(* IEC 61131-3 sources: eCockpitGit/test_project/src/%F%00 Library/%F%Common Functions/%F%Linearsation/%F%DINT, 3 files *)

(* ---- %POU%FU_diLinear2Ends.st ---- *)
//This function, converts an x, value to an y value using and 2 points on the x and y scale
//This function has ends, which means the output is never greater or smaller than the range of y
// +-----------+----------+----------+-----------------------------------------------------------------------------------------------------------------------+
// |**Version**|**Author**| **Date** |**Changes**                                                                                                            |
// +-----------+----------+----------+-----------------------------------------------------------------------------------------------------------------------+
// | 1         | NSN      | 10-12-18 | Creation                                                                                                              |
// +-----------+----------+----------+-----------------------------------------------------------------------------------------------------------------------+
FUNCTION FU_diLinear2Ends : DINT
VAR_INPUT
	XIn		:DINT;
	X1		:DINT;
	X2		:DINT;
	Y1		:DINT;
	Y2		:DINT;
END_VAR
VAR
	a		:REAL;
	b		:REAL;
END_VAR
(*%!%__DELIMITER__%!%*)
IF X2 > X1 THEN
	IF XIn <= X1 THEN	//When input is out of bounds
		FU_diLinear2Ends 			:=		Y1;
	ELSIF XIn >= X2 THEN	//When input is out of bounds
		FU_diLinear2Ends 			:=		Y2;
	ELSIF XIn > X1 AND XIn < X2 THEN	//When input is with the
		//a value is calculated
		IF X2 - X1 = 0 THEN	a := 0; ELSE a := TO_REAL(Y2 - Y1) / TO_REAL(X2 - X1); END_IF
		//b value is calculated
		b 							:=		TO_REAL(Y1) - (a * TO_REAL(X1));
		//Output is calculated
		FU_diLinear2Ends 			:=		TO_INT(a * TO_REAL (XIn) + b);
	END_IF
ELSE
	IF XIn >= X1 THEN
		FU_diLinear2Ends 			:=		Y1;
	ELSIF XIn <= X2 THEN
		FU_diLinear2Ends 			:=		Y2;
	ELSIF XIn < X1 AND XIn > X2 THEN
		//a value is calculated
		IF X2 - X1 = 0 THEN	a := 0; ELSE a := TO_REAL(Y2 - Y1) / TO_REAL(X2 - X1); END_IF
		//b value is calculated
		b 							:=		TO_REAL(Y1) - (a * TO_REAL(X1));
		//Output is calculated
		FU_diLinear2Ends 			:=		TO_INT(a * TO_REAL (XIn) + b);
	END_IF
END_IF

(* ---- %POU%FU_diLinear4Ends.st ---- *)
//This function, converts an x, value to an y value using and 3 points on the x and y scale
//This function has ends, which means the output is never greater or smaller than the range of y
// +-----------+----------+----------+-----------------------------------------------------------------------------------------------------------------------+
// |**Version**|**Author**| **Date** |**Changes**                                                                                                            |
// +-----------+----------+----------+-----------------------------------------------------------------------------------------------------------------------+
// | 1         | NSN      | 11-12-18 | Creation                                                                                                              |
// +-----------+----------+----------+-----------------------------------------------------------------------------------------------------------------------+
FUNCTION FU_diLinear4Ends : DINT
VAR_INPUT
	XIn		:DINT;
	X1		:DINT;
	X2		:DINT;
	X3		:DINT;
	X4		:DINT;
	Y1		:DINT;
	Y2		:DINT;
	Y3		:DINT;
	Y4		:DINT;
END_VAR
VAR
	a		:REAL;
	b		:REAL;
END_VAR
(*%!%__DELIMITER__%!%*)
IF X4 > X1 THEN
	IF XIn <= X1 THEN	//When input is out of bounds
		FU_diLinear4Ends 			:=		Y1;
	ELSIF XIn >= X4 THEN	//When input is out of bounds
		FU_diLinear4Ends 			:=		Y4;
	ELSIF XIn > X1 AND XIn <= X2 THEN	//When input is with the
		//a value is calculated
		IF X2 - X1 = 0 THEN	a := 0; ELSE a := TO_REAL(Y2 - Y1) / TO_REAL(X2 - X1); END_IF
		//b value is calculated
		b 							:=		TO_REAL(Y1) - (a * TO_REAL(X1));
		//Output is calculated
		FU_diLinear4Ends 			:=		TO_DINT(a * TO_REAL (XIn) + b);
	ELSIF XIn > X2 AND XIn <= X3 THEN
		//a value is calculated
		IF X3 - X2 = 0 THEN	a := 0; ELSE a := TO_REAL(Y3 - Y2) / TO_REAL(X3 - X2); END_IF
		//b value is calculated
		b 							:=		TO_REAL(Y2) - (a * TO_REAL(X2));
		//Output is calculated
		FU_diLinear4Ends 			:=		TO_INT(a * TO_REAL (XIn) + b);
	ELSIF XIn > X3 AND XIn < X4 THEN
		//a value is calculated
		IF X4 - X3 = 0 THEN	a := 0; ELSE a := TO_REAL(Y4 - Y3) / TO_REAL(X4 - X3); END_IF
		//b value is calculated
		b 							:=		TO_REAL(Y3) - (a * TO_REAL(X3));
		//Output is calculated
		FU_diLinear4Ends 			:=		TO_INT(a * TO_REAL (XIn) + b);
	END_IF
ELSE
	IF XIn >= X1 THEN
		FU_diLinear4Ends 			:=		Y1;
	ELSIF XIn <= X4 THEN
		FU_diLinear4Ends 			:=		Y4;
	ELSIF XIn < X1 AND XIn >= X2 THEN
		//a value is calculated
		IF X2 - X1 = 0 THEN	a := 0; ELSE a := TO_REAL(Y2 - Y1) / TO_REAL(X2 - X1); END_IF
		//b value is calculated
		b 							:=		TO_REAL(Y1) - (a * TO_REAL(X1));
		//Output is calculated
		FU_diLinear4Ends 			:=		TO_INT(a * TO_REAL (XIn) + b);
	ELSIF XIn < X2 AND XIn >= X3 THEN
		//a value is calculated
		IF X3 - X2 = 0 THEN	a := 0; ELSE a := TO_REAL(Y3 - Y2) / TO_REAL(X3 - X2); END_IF
		//b value is calculated
		b 							:=		TO_REAL(Y2) - (a * TO_REAL(X2));
		//Output is calculated
		FU_diLinear4Ends 			:=		TO_INT(a * TO_REAL (XIn) + b);
	ELSIF XIn < X3 AND XIn > X4 THEN
		//a value is calculated
		IF X4 - X3 = 0 THEN	a := 0; ELSE a := TO_REAL(Y4 - Y3) / TO_REAL(X4 - X3); END_IF
		//b value is calculated
		b 							:=		TO_REAL(Y3) - (a * TO_REAL(X3));
		//Output is calculated
		FU_diLinear4Ends 			:=		TO_INT(a * TO_REAL (XIn) + b);
	END_IF
END_IF

(* ---- %POU%FU_diLinearXEnds.st ---- *)
//This function, converts an x, value to an y value using and x amount of points on the x and y scale
//This function has ends, which means the output is never greater or smaller than the range of y
// |**Version**|**Author**| **Date** |**Changes**
// | 1         | NSN      | 03-01-18 | Creation
FUNCTION FU_diLinearXEnds : DINT
VAR_INPUT
	xIn			:DINT;				//Input value to be linearised
	pXArray		:POINTER TO DINT;	//Address of x array
	pYArray		:POINTER TO DINT; 	//Address of y array
	uiSize		:UINT;				//Amount of points in
END_VAR
VAR
	LowerLimit	:BOOL;
	UpperLimit	:BOOL;
	UpperXAdr	:POINTER TO DINT;	//Buffer for current x address
	LowerXAdr	:POINTER TO DINT;	//Buffer for current x address
	UpperYAdr	:POINTER TO DINT; 	//Buffer for current y address
	LowerYAdr	:POINTER TO DINT; 	//Buffer for current y address
	FOR1		:UINT;
	a			:REAL;
	b			:REAL;
	d			:BOOL;
END_VAR
(*%!%__DELIMITER__%!%*)
IF uiSize > 1 THEN
	//Direction is found
	UpperXAdr					:=		pXArray + 4;
	d							:=		UpperXAdr^ > pXArray^;

	//Pointers are set
	UpperXAdr					:=		pXArray;
	UpperYAdr					:=		pYArray;

	FOR FOR1 := 1 TO uiSize DO
		IF d THEN
			IF UpperXAdr^ <= xIn THEN
				IF FOR1 = uiSize AND UpperXAdr^ <> xIn THEN
					UpperLimit	:=		TRUE;
				ELSIF FOR1 <> uiSize THEN
					UpperXAdr	:=		UpperXAdr + 4;
					UpperYAdr	:=		UpperYAdr + 4;
				END_IF
			ELSE
				IF pXArray = UpperXAdr THEN
					LowerLimit	:=		TRUE;
				ELSE
					LowerXAdr	:=		UpperXAdr - 4;
					LowerYAdr	:=		UpperYAdr - 4;
				END_IF
				Exit;
			END_IF
		ELSE
			IF UpperXAdr^ >= xIn THEN
				IF FOR1 = uiSize AND UpperXAdr^ <> xIn THEN
					UpperLimit	:=		TRUE;
				ELSIF FOR1 <> uiSize THEN
					UpperXAdr	:=		UpperXAdr + 4;
					UpperYAdr	:=		UpperYAdr + 4;
				END_IF
			ELSE
				IF pXArray = UpperXAdr THEN
					LowerLimit	:=		TRUE;
				ELSE
					LowerXAdr	:=		UpperXAdr - 4;
					LowerYAdr	:=		UpperYAdr - 4;
				END_IF
				Exit;
			END_IF
		END_IF
	END_FOR

	IF LowerLimit THEN
		FU_diLinearXEnds			:=		pYArray^;
	ELSIF UpperLimit THEN
		FU_diLinearXEnds			:=		UpperYAdr^;
	ELSE
		IF xIn = UpperXAdr^ THEN
			FU_diLinearXEnds		:=		UpperYAdr^;
		ELSIF xIn = LowerXAdr^ THEN
			FU_diLinearXEnds		:=		LowerYAdr^;
		ELSE
			IF UpperXAdr^ - LowerXAdr^ = 0 THEN
				a				:=		0;
			ELSE
				a				:=		TO_REAL(UpperYAdr^ - LowerYAdr^) / TO_REAL(UpperXAdr^ - LowerXAdr^);
			END_IF
			b					:=		TO_REAL(LowerYAdr^) - (a * TO_REAL(LowerXAdr^));
			FU_diLinearXEnds 	:=		TO_INT(a * TO_REAL(xIn) + b);
		END_IF
	END_IF
END_IF
